PROGRAM MAIN
VAR
	fb_TimeStamp 	: FB_UpdateTimeStamp ();
	bLog_Flag		: BOOL;
	LogProcess		: LOGGINg;
END_VAR

fb_TimeStamp();

IF bLog_Flag THEN
	LogProcess( sLogEvent	 := MSG.EVENT_PROCESS, 
	 			sLogComp	 := MSG.COMP_CYLINDER_1, 
	 			sLogAction	 := MSG.ACTION_EXTEND, 
	 			sLogStatus	 := MSG.STATUS_DONE,
	 		 	blogFlag	 := TRUE);
	IF LogProcess.blog_complete OR LogProcess.blog_error THEN
		bLog_Flag 			:= FALSE;
	END_IF
END_IF

END_PROGRAM

(* stored: Version 1.1.0.1, ProductVersion 3.1.4024.12
   POU MAIN: Id {adb1c04d-0f03-4f01-b08b-c18b8d85a7bd}, SpecialFunc None *)
